TYPE E_XML_WritingMode :
(
	E_CS_HEADER,
	E_OUTER_HEADER,
	E_PACK_ITEM,
	E_OUTER_ENDING,
	E_CS_ENDING
);
END_TYPE

(* stored: Version 1.1.0.1, ProductVersion 3.1.4024.15
   DUT E_XML_WritingMode: Id {4da77ace-f487-4925-a917-6d5215984c4d} *)
